(* IEC 61131-3 sources: ArfBotOS/Codesys-4/ArfBotOS.fbsdev/Application.iecapp^/FUN/FB_ProgramProcessor.fb.st^/protected, 9 files *)

(* ---- M_Aborting.meth.st ---- *)
METHOD PROTECTED M_Aborting : BOOL

CASE _SeqAborting OF
	0:
		_ProcessCommands.M_Abort();
		_SeqAborting := _SeqAborting + 1;
	1:
		IF _ProcessCommands.PropCurrentState = PACK_ML.State.Aborted THEN
			_SeqAborting := 0;
			SUPER^.M_StateComplete();
		END_IF

END_CASE

(*IF ItfActiveModule <> 0 THEN
	ItfActiveModule.M_Abort();
	IF ItfActiveModule.PropCurrentState = PACK_ML.State.Aborted THEN
		SUPER^.M_StateComplete();
	END_IF
ELSE
	SUPER^.M_StateComplete();
END_IF*)
END_METHOD

(* ---- M_Clearing.meth.st ---- *)
METHOD PROTECTED M_Clearing : BOOL

SUPER^.M_StateComplete();

(*IF SUPER^.Flags[GVL_App.HOME_COMPLETE].Value THEN
	CASE _SeqClearing OF
		0:
			_ProcessMoveCommand.M_Home();
			_SeqClearing := _SeqClearing + 1;
		1:
			IF _ProcessMoveCommand.PropCurrentState = PACK_ML.State.Idle THEN
				_SeqClearing := _SeqClearing + 1;
			END_IF
		2:
			IF NOT _ProcessMoveCommand.Error THEN
				_ProcessMoveCommand.Command := GVL_App.Pose2;
				_ProcessMoveCommand.M_Start();
				_SeqClearing := _SeqClearing + 1;
			ELSE
				SUPER^._M_Error(Description:='Move processor errored. Please reset and try again');
				_SeqClearing := -1;
			END_IF
		3:
			IF _ProcessMoveCommand.PropCurrentState = PACK_ML.State.Execute THEN
				_SeqClearing := _SeqClearing + 1;
			END_IF
		4:
			IF _ProcessMoveCommand.PropCurrentState = PACK_ML.State.Complete
				OR _ProcessMoveCommand.PropCurrentState = PACK_ML.State.Stopped
				OR _ProcessMoveCommand.PropCurrentState = PACK_ML.State.Aborted
				OR _ProcessMoveCommand.PropCurrentState = PACK_ML.State.Idle  THEN
					SUPER^.M_StateComplete();
					_SeqClearing := 0;
			END_IF
	END_CASE
ELSE
	SUPER^._M_Error(Description:='Drives are not homed. Please home and try again');
	_SeqClearing := -1;
END_IF

IF _ProcessMoveCommand.Error THEN
	SUPER^._M_Error(Description:='Move processor in error state. Please reset and try again');
	_SeqClearing := -1;
END_IF
*)

(*
IF ItfActiveModule <> 0 THEN
	//
	CASE _Seq OF
		0:
			IF NOT ItfActiveModule.PropCurrentState = PACK_ML.State.Stopped THEN
				ItfActiveModule.M_Abort();
				_Seq := 1;
			ELSE
				SUPER^.M_StateComplete();
			END_IF
		1:
			CASE ItfActiveModule.PropCurrentState OF
				PACK_ML.State.Aborted:
					ItfActiveModule.Clear();
				PACK_ML.State.Stopped:
					_Seq := 0;
			END_CASE

	END_CASE
ELSE
	_Seq := 0;
	SUPER^.M_StateComplete();
END_IF
*)
END_METHOD

(* ---- M_Execute.meth.st ---- *)
METHOD PROTECTED M_Execute : BOOL
VAR
    _ErrorDescription: STRING;
END_VAR

{warning disable C0371}
// here we want to execute our commands/jobs/etc and set completed when done.
//
CASE _SeqMain OF
  	_STEP_DONE:
		_SeqMain := _STEP_IDLE;

	_STEP_IDLE:
		// hang out here until called to run
		_CurrentPrgIdx := 0;
		SUPER^.M_StateComplete();

	_STEP_PRG: //
		IF NOT Enable THEN
			_SeqMain := _STEP_DONE;
            IF NOT GVL_App.Enable THEN
                _ErrorDescription := 'Robot not enabled';
            END_IF
            IF NOT PersistentVars.Flags[GVL_App.HOME_COMPLETE].Value THEN
                _ErrorDescription := CONCAT(_ErrorDescription, ' | Robot not homed');
            END_IF
            IF GVL_App.xActiveAlarm THEN
                _ErrorDescription := CONCAT(_ErrorDescription, ' | Active alarms exist');
            END_IF
            IF _ErrorDescription = '' THEN
                _ErrorDescription := 'Not enabled';
            END_IF
            _M_Error(Description := _ErrorDescription);

		ELSIF _CurrentPrgIdx <= GVL_App.PROG_ARR_END AND _CurrentPrgIdx >= GVL_App.PROG_ARR_BEG THEN
			//
			StatusText := '';
			ItfActiveModule := _ProcessCommands;
			ItfActiveProcessorUnitMode := _ProcessCommands.ItfUnitMode;

			IF _ProcessCommands.M_SetCommands(StartingCommand:=0, Commands:=Programs[_CurrentPrgIdx].Commands) THEN
				_ProcessCommands.M_Start();
				_SeqMain := _STEP_WAIT_EXECUTE;
			ELSE
				SUPER^.M_Error('Failed to set Command Processor. Check commands.');
				_SeqMain := _STEP_ERR;
			END_IF

		ELSE
			_SeqMain := _STEP_DONE;
		END_IF

	_STEP_WAIT_EXECUTE:
		IF _ProcessCommands.PropCurrentState = PACK_ML.State.Execute THEN
			_SeqMain := _STEP_WAIT_IDLE;
		END_IF

	_STEP_WAIT_IDLE: // wait for program to finish
		//
		IF _ProcessCommands.PropCurrentState = PACK_ML.State.Idle THEN
			IF _Returning[_CurrentPrgIdx] THEN
				_Returning[_CurrentPrgIdx] := FALSE;
				IF _ReturnPrograms[_CurrentPrgIdx] <= GVL_App.PROG_ARR_END AND_THEN _ReturnPrograms[_CurrentPrgIdx] >= GVL_App.PROG_ARR_BEG
					AND_THEN _ReturnCommands[_CurrentPrgIdx] <= GVL_App.PROG_CMDS_ARR_END + 1 AND_THEN _ReturnCommands[_CurrentPrgIdx] >= GVL_App.PROG_CMDS_ARR_BEG // +1 because we want to be able to tell if calling program was on last command
					THEN
						//
						IF _ProcessCommands.M_SetCommands(StartingCommand:=_ReturnCommands[_CurrentPrgIdx], Commands:=Programs[_ReturnPrograms[_CurrentPrgIdx]].Commands) THEN
							_CurrentPrgIdx := _ReturnPrograms[_CurrentPrgIdx];
							_ProcessCommands.M_Start();
							_SeqMain := _STEP_WAIT_EXECUTE;
						ELSE
							SUPER^.M_Error('Failed to set Command Processor. Check commands.');
							_SeqMain := _STEP_ERR;
						END_IF
				ELSE
					_SeqMain := _STEP_DONE;
				END_IF
			ELSE
				_SeqMain := _STEP_DONE;
			END_IF
		END_IF
		//
		IF _ProcessCommands.PropError THEN
			SUPER^._UnitMode.Suspend();
			_SeqMain := _STEP_ERR;
		END_IF

	_STEP_ERR: //

END_CASE

// watch for rising edge of idle state. this was done for all processors since
// the vision processor runs in a separate task and isnt guaranteed to start in the same
// PLC scan.
//_ProcessorDoneRtrig(clk:=ItfActiveProcessorUnitMode.CurrentState = PACK_ML.State.Idle);
{warning restore C0371}
END_METHOD

(* ---- M_Idle.meth.st ---- *)
METHOD PROTECTED M_Idle : BOOL

// in this state, we want to reset all the function blocks and hang out
FOR _i:=GVL_App.PROG_ARR_BEG TO GVL_App.PROG_ARR_END BY 1 DO
	_Returning[_i] := FALSE;
END_FOR
(*FOR _i:=GVL_App.PROG_ARR_BEG TO GVL_App.PROG_ARR_END BY 1 DO
	_ReturnPrograms[_i] := 0;
END_FOR
FOR _i:=GVL_App.PROG_CMDS_ARR_BEG TO GVL_App.PROG_CMDS_ARR_END BY 1 DO
	_ReturnCommands[_i] := 0;
END_FOR*)
_SeqMain := _STEP_IDLE;
_SeqAborting := 0;
_SeqClearing := 0;
_SeqResetting := 0;
END_METHOD

(* ---- M_Resetting.meth.st ---- *)
METHOD PROTECTED M_Resetting : BOOL

CASE _SeqResetting OF
	0:
		_ProcessCommands.M_Home();
		_SeqResetting := _SeqResetting + 1;
	1:
		IF _ProcessCommands.PropCurrentState = PACK_ML.State.Idle THEN
			_SeqResetting := 0;
			SUPER^.M_StateComplete();
		END_IF

END_CASE

SUPER^.M_Reset();

(*IF ItfActiveModule <> 0 THEN
	CASE _Seq OF
		0:
			IF NOT ItfActiveModule.PropCurrentState = PACK_ML.State.Idle THEN
				ItfActiveModule.M_Home();
				_Seq := 1;
			ELSE
				SUPER^.M_StateComplete();
			END_IF
		1:
			IF ItfActiveModule.PropCurrentState = PACK_ML.State.Idle THEN
				_Seq := 0;
			END_IF

	END_CASE

ELSE
	SUPER^.M_StateComplete();
	_Seq := 0;

END_IF*)
END_METHOD

(* ---- M_SetPackML.meth.st ---- *)
METHOD PROTECTED M_SetPackML : BOOL

// SUPER already does this but the default is eInitialState:=PACK_ML.State.Idle
// and we want PACK_ML.State.Aborted for the Orchestrator
SUPER^._UnitMode(sName := 'Program Processor',
				eInitialState := PACK_ML.State.Aborted,
				xActive := TRUE);
END_METHOD

(* ---- M_Starting.meth.st ---- *)
METHOD PROTECTED M_Starting : BOOL

// here we want to clear things and get ready for the execute state
// we can consider this the "INIT" state
(*FOR _i:=GVL_App.PROG_ARR_BEG TO GVL_App.PROG_ARR_END BY 1 DO
	_Returning[_i] := FALSE;
END_FOR
FOR _i:=GVL_App.PROG_ARR_BEG TO GVL_App.PROG_ARR_END BY 1 DO
	_ReturnPrograms[_i] := 0;
END_FOR
FOR _i:=GVL_App.PROG_CMDS_ARR_BEG TO GVL_App.PROG_CMDS_ARR_END BY 1 DO
	_ReturnCommands[_i] := 0;
END_FOR*)
//_CurrentPrgIdx := 0;
_SeqMain := _STEP_PRG;
SUPER^.M_StateComplete();
END_METHOD

(* ---- M_UnHolding.meth.st ---- *)
METHOD PROTECTED M_Unholding : BOOL

//
IF ItfActiveModule <> 0 THEN
	ItfActiveModule.M_Start();
	IF ItfActiveModule.PropCurrentState = PACK_ML.State.Execute THEN
		SUPER^.M_StateComplete();
	END_IF

ELSE
	SUPER^.M_StateComplete();

END_IF

//
_SeqMain := _STEP_WAIT_IDLE;
END_METHOD

(* ---- M_UnSuspending.meth.st ---- *)
METHOD PROTECTED M_UnSuspending : BOOL

//
IF ItfActiveModule <> 0 THEN
	ItfActiveModule.M_Start();
	IF ItfActiveModule.PropCurrentState = PACK_ML.State.Execute THEN
		SUPER^.M_StateComplete();
	END_IF

ELSE
	SUPER^.M_StateComplete();

END_IF

//
_SeqMain := _STEP_WAIT_IDLE;
END_METHOD
